% RSLogix 500 project HANDS ON TEST 1.RSS, saved by version 10.00.00.00 %
PROJECT "UNTITLED"    % processor: Bul.1763 MicroLogix 1100 Series B %

PROGRAM FILES
  LAD 2   6 rungs

DATA FILES
  O0 OUTPUT  4 elements
  I1 INPUT  6 elements
  S2 STATUS  66 elements
  B3 BINARY  1 elements
  T4 TIMER  1 elements
  C5 COUNTER  1 elements
  R6 CONTROL  1 elements
  N7 INTEGER  1 elements
  F8 FLOAT  1 elements

LADDER 2
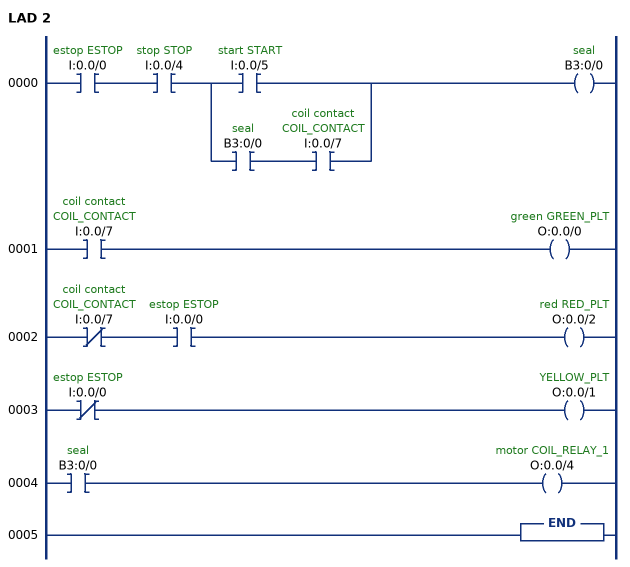
% Rung: 0 %
SOR XIC I:0.0/0 XIC I:0.0/4 BST XIC I:0.0/5 NXB XIC B3:0/0 XIC I:0.0/7 BND OTE B3:0/0 EOR
%   I:0.0/0  ESTOP  "estop" %
%   I:0.0/4  STOP  "stop" %
%   I:0.0/5  START  "start" %
%   B3:0/0  "seal" %
%   I:0.0/7  COIL_CONTACT  "coil contact" %
% Rung: 1 %
SOR XIC I:0.0/7 OTE O:0.0/0 EOR
%   I:0.0/7  COIL_CONTACT  "coil contact" %
%   O:0.0/0  GREEN_PLT  "green" %
% Rung: 2 %
SOR XIO I:0.0/7 XIC I:0.0/0 OTE O:0.0/2 EOR
%   I:0.0/7  COIL_CONTACT  "coil contact" %
%   I:0.0/0  ESTOP  "estop" %
%   O:0.0/2  RED_PLT  "red" %
% Rung: 3 %
SOR XIO I:0.0/0 OTE O:0.0/1 EOR
%   I:0.0/0  ESTOP  "estop" %
%   O:0.0/1  YELLOW_PLT %
% Rung: 4 %
SOR XIC B3:0/0 OTE O:0.0/4 EOR
%   B3:0/0  "seal" %
%   O:0.0/4  COIL_RELAY_1  "motor" %
% Rung: 5 %
SOR END EOR

OTHER DOCUMENTED ADDRESSES
  B30:0/0  B
  I:0.0/1  3POS_SS  "THREE POSITION SWITCH"
  I:0.0/2  3POS_SSB  "POSITION B"
  I:0.0/3  2POS_SS  "2 POSITION SELECTOR SWITCH A ONLY"
  I:0.0/6  PB_NO  "PBNO"
  I:0.0/8  COIL_CONTACT8_6  "RELAY CONTACT 8 6"
  I:0.0/9  MS_CONTACTS_NO  "MOTOR STARTER CONTACTS"
  O:0.0/3  BLUE_PLT
